PROGRAM INTERNAL FsP_CorePlayground
VAR
	fbObj : FsFB_Object;
	Sz0,Sz1 : FsT_Size;
	sName : STRING(255);
	arData : ARRAY[0..3] OF FsT_LStr;
END_VAR

arData[0] := fbObj.InstancePath;
arData[1] := fbObj.TypeName;
arData[2] := FsF_GetVariablePathByAddress(ADR(fbObj), SIZEOF(fbObj));
Sz0 := fbObj.Size;

END_PROGRAM

(* stored: Version 1.1.0.1, ProductVersion 3.1.4024.4
   POU FsP_CorePlayground: Id {fe32e6f4-2a42-43f5-bef2-f3cbb688e3ff}, SpecialFunc None *)
